INTERFACE I_TankController

METHOD ApplyCooling 
VAR_INPUT
END_VAR
END_METHOD

METHOD CheckSafety : BOOL
VAR_INPUT
END_VAR
END_METHOD

END_INTERFACE

(* stored: Version 1.1.0.1, ProductVersion 3.1.4024.16
   Itf I_TankController: Id {694224f3-b411-404f-9f19-e17cb45067f5}
   Method ApplyCooling: Id {2d1b7223-85f0-478d-b4dc-b663201c99cf}
   Method CheckSafety: Id {46370de7-60ed-4e93-bcd4-01bbd698d84c} *)
